{attribute 'GeneratedUsingTerminal: EL3692-0000-0017'}
{attribute addProperty BoxType "EL3692-0000-0017"}
{attribute addProperty Id "SAI_Inputs_Channel_1AT %I*SAI_Inputs_Channel_9DCD655714SAI_Range_Channel_1AT %I*SAI_Range_Channel_BDBF6DA92SAI_Inputs_Real_Channel_1AT %I*SAI_Inputs_Real_Channel_CCECF13D4SAI_Inputs_Channel_2AT %I*SAI_Inputs_Channel_9DCD655714SAI_Range_Channel_2AT %I*SAI_Range_Channel_BDBF6DA92SAI_Inputs_Real_Channel_2AT %I*SAI_Inputs_Real_Channel_CCECF13D4WcStateAT %I*WcState_9091E0EB2InfoDataAT %I*InfoData_94A18F5E2"}
{attribute addProperty CRC "3502871"}
{attribute addProperty Size "44"}
TYPE EL3692_00357317 EXTENDS EtcSlaveTerminalBase_947E5A46 :
STRUCT
	{attribute addProperty Name "SAI_Inputs_Channel_1"}
	SAI_Inputs_Channel_1 : SAI_Inputs_Channel_9DCD6557;
	{attribute addProperty Name "SAI_Range_Channel_1"}
	SAI_Range_Channel_1 : SAI_Range_Channel_BDBF6DA9;
	{attribute addProperty Name "SAI_Inputs_Real_Channel_1"}
	SAI_Inputs_Real_Channel_1 : SAI_Inputs_Real_Channel_CCECF13D;
	{attribute addProperty Name "SAI_Inputs_Channel_2"}
	SAI_Inputs_Channel_2 : SAI_Inputs_Channel_9DCD6557;
	{attribute addProperty Name "SAI_Range_Channel_2"}
	SAI_Range_Channel_2 : SAI_Range_Channel_BDBF6DA9;
	{attribute addProperty Name "SAI_Inputs_Real_Channel_2"}
	SAI_Inputs_Real_Channel_2 : SAI_Inputs_Real_Channel_CCECF13D;
	{attribute addProperty Name "WcState"}
	WcState : WcState_9091E0EB;
	{attribute addProperty Name "InfoData"}
	InfoData : InfoData_94A18F5E;
END_STRUCT
END_TYPE

(* stored: Version 1.2.0.0, ProductVersion 3.1.4024.9
   DUT EL3692_00357317: Id {3c0ec7c0-0b9f-4c47-82cf-9685a6c1137c} *)
